ABB RAPID module: Module1.mod

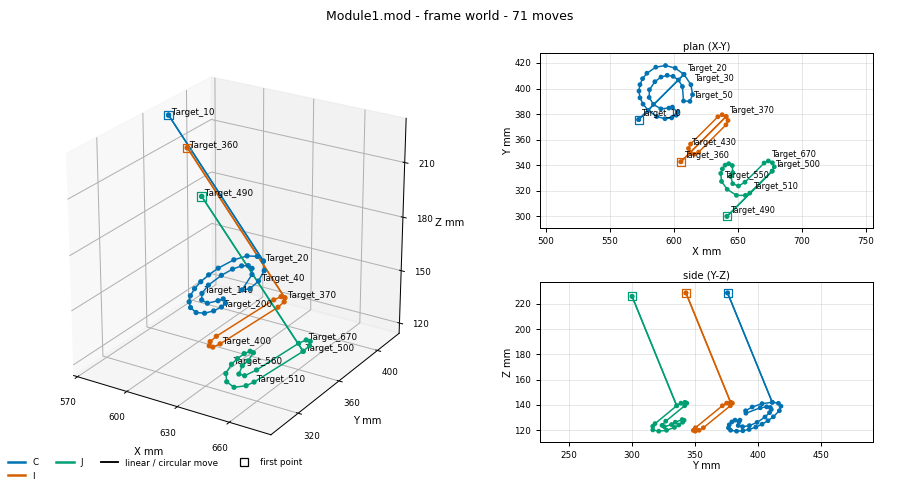
[picture p0: tool path of Module1.mod in frame world, 71 of 73 moves have a stored position in this frame; points joined in program order, loops and branches not executed]
MODULE Module1
        CONST robtarget Target_10:=[[103.793570023,149.495277511,99.999575997],[0.000000083,-0.533161025,0.846013783,0.00000013],[0,0,0,0],[9E+09,9E+09,9E+09,9E+09,9E+09,9E+09]];
    CONST robtarget Target_20:=[[103.793570137,149.495246706,-0.000424002],[0.000000083,-0.533161025,0.846013783,0.00000013],[0,0,-1,0],[9E+09,9E+09,9E+09,9E+09,9E+09,9E+09]];
    CONST robtarget Target_30:=[[113.359124829,147.348233514,-0.000423331],[0.000000133,-0.533160983,0.846013809,0.000000079],[0,0,-1,0],[9E+09,9E+09,9E+09,9E+09,9E+09,9E+09]];
    CONST robtarget Target_40:=[[119.782709001,142.041794411,-0.000421688],[0.000000153,-0.533160941,0.846013836,0.000000008],[0,0,-1,0],[9E+09,9E+09,9E+09,9E+09,9E+09,9E+09]];
    CONST robtarget Target_50:=[[122.016999147,136.089505814,-0.000419852],[-0.000000082,-0.533160946,0.846013833,-0.00000013],[0,0,-1,0],[9E+09,9E+09,9E+09,9E+09,9E+09,9E+09]];
    CONST robtarget Target_60:=[[118.316456088,132.214408841,-0.000418663],[-0.000000081,-0.533160946,0.846013833,-0.000000131],[0,0,-1,0],[9E+09,9E+09,9E+09,9E+09,9E+09,9E+09]];
    CONST robtarget Target_70:=[[109.693492554,140.750095424,-0.000421301],[-0.000000082,-0.533160946,0.846013833,-0.000000131],[0,0,-1,0],[9E+09,9E+09,9E+09,9E+09,9E+09,9E+09]];
    CONST robtarget Target_80:=[[103.863391701,142.373446861,-0.000421809],[-0.000000081,-0.533160946,0.846013833,-0.000000131],[0,0,-1,0],[9E+09,9E+09,9E+09,9E+09,9E+09,9E+09]];
    CONST robtarget Target_90:=[[98.906060436,141.326123357,-0.000421492],[-0.000000081,-0.533160946,0.846013833,-0.000000131],[0,0,-1,0],[9E+09,9E+09,9E+09,9E+09,9E+09,9E+09]];
    CONST robtarget Target_100:=[[95.065874244,138.184152838,-0.000420528],[-0.000000082,-0.533160946,0.846013833,-0.000000131],[0,0,-1,0],[9E+09,9E+09,9E+09,9E+09,9E+09,9E+09]];
    CONST robtarget Target_110:=[[92.604664001,133.104633832,-0.000418965],[-0.000000082,-0.533160946,0.846013833,-0.000000131],[0,0,-1,0],[9E+09,9E+09,9E+09,9E+09,9E+09,9E+09]];
    CONST robtarget Target_120:=[[91.784260586,126.244664864,-0.000416854],[-0.000000082,-0.533160946,0.846013833,-0.00000013],[0,0,-1,0],[9E+09,9E+09,9E+09,9E+09,9E+09,9E+09]];
    CONST robtarget Target_130:=[[93.2330581,117.656612109,-0.000414207],[0.000000152,-0.533160925,0.846013846,-0.000000026],[0,0,-1,0],[9E+09,9E+09,9E+09,9E+09,9E+09,9E+09]];
    CONST robtarget Target_140:=[[97.335075165,112.542182317,-0.000412627],[0.00000014,-0.533160974,0.846013815,0.000000065],[0,0,-1,0],[9E+09,9E+09,9E+09,9E+09,9E+09,9E+09]];
    CONST robtarget Target_150:=[[103.549194637,110.849009312,-0.000412097],[0.000000083,-0.533161025,0.846013783,0.00000013],[0,0,-1,0],[9E+09,9E+09,9E+09,9E+09,9E+09,9E+09]];
    CONST robtarget Target_160:=[[110.094966554,112.769102406,-0.000412682],[-0.000000009,-0.533161065,0.846013758,0.000000153],[0,0,-1,0],[9E+09,9E+09,9E+09,9E+09,9E+09,9E+09]];
    CONST robtarget Target_170:=[[114.127162057,118.389738556,-0.000414408],[-0.000000094,-0.533161077,0.846013751,0.000000123],[0,0,-1,0],[9E+09,9E+09,9E+09,9E+09,9E+09,9E+09]];
    CONST robtarget Target_180:=[[115.5235934,121.252422806,-0.000415289],[-0.000000055,-0.533161075,0.846013751,0.000000144],[0,0,-1,0],[9E+09,9E+09,9E+09,9E+09,9E+09,9E+09]];
    CONST robtarget Target_190:=[[120.987131026,121.252422805,-0.000415283],[0.00000015,-0.533160956,0.846013827,0.000000034],[0,0,-1,0],[9E+09,9E+09,9E+09,9E+09,9E+09,9E+09]];
    CONST robtarget Target_200:=[[122.12173149,118.45956012,-0.000414421],[-0.000000082,-0.533160946,0.846013833,-0.00000013],[0,0,-1,0],[9E+09,9E+09,9E+09,9E+09,9E+09,9E+09]];
    CONST robtarget Target_210:=[[121.091863374,113.886247475,-0.000413014],[-0.000000082,-0.533160946,0.846013833,-0.000000131],[0,0,-1,0],[9E+09,9E+09,9E+09,9E+09,9E+09,9E+09]];
    CONST robtarget Target_220:=[[117.82770511,109.068559346,-0.000411533],[-0.000000081,-0.533160946,0.846013833,-0.00000013],[0,0,-1,0],[9E+09,9E+09,9E+09,9E+09,9E+09,9E+09]];
    CONST robtarget Target_230:=[[112.119791998,105.210917765,-0.000410351],[-0.000000081,-0.533160946,0.846013833,-0.000000131],[0,0,-1,0],[9E+09,9E+09,9E+09,9E+09,9E+09,9E+09]];
    CONST robtarget Target_240:=[[104.037945604,103.727209468,-0.000409903],[-0.000000081,-0.533160946,0.846013833,-0.000000131],[0,0,-1,0],[9E+09,9E+09,9E+09,9E+09,9E+09,9E+09]];
    CONST robtarget Target_250:=[[97.666727605,104.390514357,-0.000410115],[-0.000000082,-0.533160946,0.846013833,-0.000000131],[0,0,-1,0],[9E+09,9E+09,9E+09,9E+09,9E+09,9E+09]];
    CONST robtarget Target_260:=[[92.447565465,106.450250589,-0.000410756],[-0.000000081,-0.533160946,0.846013833,-0.000000131],[0,0,-1,0],[9E+09,9E+09,9E+09,9E+09,9E+09,9E+09]];
    CONST robtarget Target_270:=[[88.15353909,110.150793647,-0.0004119],[-0.000000082,-0.533160946,0.846013833,-0.000000132],[0,0,-1,0],[9E+09,9E+09,9E+09,9E+09,9E+09,9E+09]];
    CONST robtarget Target_280:=[[85.168667098,114.828838645,-0.000413345],[-0.000000082,-0.533160947,0.846013833,-0.00000013],[0,0,-1,0],[9E+09,9E+09,9E+09,9E+09,9E+09,9E+09]];
    CONST robtarget Target_290:=[[83.318395571,120.327287055,-0.000415041],[-0.000000082,-0.533160946,0.846013833,-0.00000013],[0,0,-1,0],[9E+09,9E+09,9E+09,9E+09,9E+09,9E+09]];
    CONST robtarget Target_300:=[[82.707456862,126.558861919,-0.000416961],[-0.00000013,-0.533161068,0.846013756,0.000000082],[0,0,-1,0],[9E+09,9E+09,9E+09,9E+09,9E+09,9E+09]];
    CONST robtarget Target_310:=[[84.260986733,136.124416613,-0.000419906],[-0.000000094,-0.533161077,0.846013751,0.000000123],[0,0,-1,0],[9E+09,9E+09,9E+09,9E+09,9E+09,9E+09]];
    CONST robtarget Target_320:=[[88.712111639,143.350948806,-0.000422127],[-0.000000037,-0.533161072,0.846013754,0.000000149],[0,0,-1,0],[9E+09,9E+09,9E+09,9E+09,9E+09,9E+09]];
    CONST robtarget Target_330:=[[95.502259042,147.924261449,-0.000423527],[0.000000028,-0.533161053,0.846013766,0.000000151],[0,0,-1,0],[9E+09,9E+09,9E+09,9E+09,9E+09,9E+09]];
    CONST robtarget Target_340:=[[103.793570137,149.495246706,-0.000424002],[0.000000083,-0.533161025,0.846013783,0.00000013],[0,0,-1,0],[9E+09,9E+09,9E+09,9E+09,9E+09,9E+09]];
    CONST robtarget Target_350:=[[103.793570023,149.495277511,99.999575997],[0.000000083,-0.533161025,0.846013783,0.00000013],[0,0,-1,0],[9E+09,9E+09,9E+09,9E+09,9E+09,9E+09]];
    CONST robtarget Target_360:=[[150.434376851,149.495277492,99.999576051],[0.000000083,-0.533161025,0.846013783,0.00000013],[0,0,0,0],[9E+09,9E+09,9E+09,9E+09,9E+09,9E+09]];
    CONST robtarget Target_370:=[[150.434376963,149.495246688,-0.000423949],[0.000000083,-0.533161025,0.846013783,0.00000013],[0,0,-1,0],[9E+09,9E+09,9E+09,9E+09,9E+09,9E+09]];
    CONST robtarget Target_380:=[[153.681079834,148.15118152,-0.000423532],[0.000000151,-0.533160952,0.846013829,0.000000028],[0,0,-1,0],[9E+09,9E+09,9E+09,9E+09,9E+09,9E+09]];
    CONST robtarget Target_390:=[[154.93786804,144.049164452,-0.000422267],[-0.000000082,-0.533160946,0.846013833,-0.00000013],[0,0,-1,0],[9E+09,9E+09,9E+09,9E+09,9E+09,9E+09]];
    CONST robtarget Target_400:=[[154.937868027,109.208202466,-0.000411535],[-0.000000082,-0.533160946,0.846013833,-0.00000013],[0,0,-1,0],[9E+09,9E+09,9E+09,9E+09,9E+09,9E+09]];
    CONST robtarget Target_410:=[[153.681079818,105.088730007,-0.000410266],[-0.000000081,-0.533160946,0.846013833,-0.000000131],[0,0,-1,0],[9E+09,9E+09,9E+09,9E+09,9E+09,9E+09]];
    CONST robtarget Target_420:=[[150.434376946,103.72720945,-0.00040985],[-0.000000081,-0.533160946,0.846013833,-0.000000131],[0,0,-1,0],[9E+09,9E+09,9E+09,9E+09,9E+09,9E+09]];
    CONST robtarget Target_430:=[[147.257495644,105.106185402,-0.000410279],[-0.000000082,-0.533160946,0.846013833,-0.000000131],[0,0,-1,0],[9E+09,9E+09,9E+09,9E+09,9E+09,9E+09]];
    CONST robtarget Target_440:=[[146.000707437,109.208202469,-0.000411544],[-0.00000013,-0.533161068,0.846013756,0.000000082],[0,0,-1,0],[9E+09,9E+09,9E+09,9E+09,9E+09,9E+09]];
    CONST robtarget Target_450:=[[146.00070745,144.049164456,-0.000422278],[-0.00000013,-0.533161068,0.846013756,0.000000082],[0,0,-1,0],[9E+09,9E+09,9E+09,9E+09,9E+09,9E+09]];
    CONST robtarget Target_460:=[[147.240040268,148.13372613,-0.000423534],[-0.000000041,-0.533161073,0.846013753,0.000000149],[0,0,-1,0],[9E+09,9E+09,9E+09,9E+09,9E+09,9E+09]];
    CONST robtarget Target_470:=[[150.434376963,149.495246688,-0.000423949],[0.000000083,-0.533161025,0.846013783,0.00000013],[0,0,-1,0],[9E+09,9E+09,9E+09,9E+09,9E+09,9E+09]];
    CONST robtarget Target_480:=[[150.434376851,149.495277492,99.999576051],[0.000000083,-0.533161025,0.846013783,0.00000013],[0,0,-1,0],[9E+09,9E+09,9E+09,9E+09,9E+09,9E+09]];
    CONST robtarget Target_490:=[[206.082165832,144.049195237,99.999577791],[-0.000000082,-0.533160946,0.846013833,-0.00000013],[0,0,0,0],[9E+09,9E+09,9E+09,9E+09,9E+09,9E+09]];
    CONST robtarget Target_500:=[[206.082165946,144.049164432,-0.000422209],[-0.000000082,-0.533160946,0.846013833,-0.00000013],[0,0,-1,0],[9E+09,9E+09,9E+09,9E+09,9E+09,9E+09]];
    CONST robtarget Target_510:=[[205.820335058,115.753974363,-0.000413492],[-0.000000082,-0.533160946,0.846013833,-0.000000131],[0,0,-1,0],[9E+09,9E+09,9E+09,9E+09,9E+09,9E+09]];
    CONST robtarget Target_520:=[[204.650823807,111.442492595,-0.000412166],[-0.000000082,-0.533160947,0.846013833,-0.00000013],[0,0,-1,0],[9E+09,9E+09,9E+09,9E+09,9E+09,9E+09]];
    CONST robtarget Target_530:=[[199.69349254,105.769490269,-0.000410425],[-0.000000082,-0.533160946,0.846013833,-0.000000131],[0,0,-1,0],[9E+09,9E+09,9E+09,9E+09,9E+09,9E+09]];
    CONST robtarget Target_540:=[[191.24508292,103.727209435,-0.000409804],[-0.000000081,-0.533160946,0.846013833,-0.000000131],[0,0,-1,0],[9E+09,9E+09,9E+09,9E+09,9E+09,9E+09]];
    CONST robtarget Target_550:=[[183.77417524,105.14109617,-0.000410249],[-0.000000081,-0.533160946,0.846013833,-0.000000131],[0,0,-1,0],[9E+09,9E+09,9E+09,9E+09,9E+09,9E+09]];
    CONST robtarget Target_560:=[[178.921576328,109.731864211,-0.000411669],[-0.000000082,-0.533160946,0.846013833,-0.000000131],[0,0,-1,0],[9E+09,9E+09,9E+09,9E+09,9E+09,9E+09]];
    CONST robtarget Target_570:=[[177.35059107,113.624416577,-0.000412869],[-0.000000081,-0.533160946,0.846013833,-0.00000013],[0,0,-1,0],[9E+09,9E+09,9E+09,9E+09,9E+09,9E+09]];
    CONST robtarget Target_580:=[[176.757107751,117.831165995,-0.000414166],[-0.00000013,-0.533161068,0.846013756,0.000000082],[0,0,-1,0],[9E+09,9E+09,9E+09,9E+09,9E+09,9E+09]];
    CONST robtarget Target_590:=[[177.926619001,121.042958082,-0.000415153],[-0.00000003,-0.533161071,0.846013754,0.000000151],[0,0,-1,0],[9E+09,9E+09,9E+09,9E+09,9E+09,9E+09]];
    CONST robtarget Target_600:=[[180.946401779,122.160103154,-0.000415494],[0.000000083,-0.533161025,0.846013783,0.00000013],[0,0,-1,0],[9E+09,9E+09,9E+09,9E+09,9E+09,9E+09]];
    CONST robtarget Target_610:=[[185.030963453,117.935898343,-0.000414188],[0.000000145,-0.533160914,0.846013853,-0.000000052],[0,0,-1,0],[9E+09,9E+09,9E+09,9E+09,9E+09,9E+09]];
    CONST robtarget Target_620:=[[186.043376174,114.235355286,-0.000413048],[0.00000015,-0.533160923,0.846013848,-0.000000032],[0,0,-1,0],[9E+09,9E+09,9E+09,9E+09,9E+09,9E+09]];
    CONST robtarget Target_630:=[[191.210172139,110.849009279,-0.000411998],[0.000000083,-0.533161025,0.846013783,0.00000013],[0,0,-1,0],[9E+09,9E+09,9E+09,9E+09,9E+09,9E+09]];
    CONST robtarget Target_640:=[[195.661297043,113.03093325,-0.000412666],[-0.000000061,-0.533161076,0.846013751,0.000000141],[0,0,-1,0],[9E+09,9E+09,9E+09,9E+09,9E+09,9E+09]];
    CONST robtarget Target_650:=[[197.145005346,119.576705165,-0.00041468],[-0.00000013,-0.533161068,0.846013756,0.000000082],[0,0,-1,0],[9E+09,9E+09,9E+09,9E+09,9E+09,9E+09]];
    CONST robtarget Target_660:=[[197.145005355,144.049164436,-0.000422219],[-0.00000013,-0.533161068,0.846013756,0.000000082],[0,0,-1,0],[9E+09,9E+09,9E+09,9E+09,9E+09,9E+09]];
    CONST robtarget Target_670:=[[198.331971998,148.133726111,-0.000423476],[-0.000000043,-0.533161074,0.846013753,0.000000148],[0,0,-1,0],[9E+09,9E+09,9E+09,9E+09,9E+09,9E+09]];
    CONST robtarget Target_680:=[[201.578674869,149.495246669,-0.000423891],[0.000000083,-0.533161025,0.846013783,0.00000013],[0,0,-1,0],[9E+09,9E+09,9E+09,9E+09,9E+09,9E+09]];
    CONST robtarget Target_690:=[[204.860288522,148.133726108,-0.000423468],[0.000000152,-0.53316095,0.84601383,0.000000025],[0,0,-1,0],[9E+09,9E+09,9E+09,9E+09,9E+09,9E+09]];
    CONST robtarget Target_700:=[[206.082165946,144.049164432,-0.000422209],[-0.000000082,-0.533160946,0.846013833,-0.00000013],[0,0,-1,0],[9E+09,9E+09,9E+09,9E+09,9E+09,9E+09]];
    CONST robtarget Target_710:=[[206.082165832,144.049195237,99.999577791],[-0.000000082,-0.533160946,0.846013833,-0.00000013],[0,0,-1,0],[9E+09,9E+09,9E+09,9E+09,9E+09,9E+09]];
    CONST jointtarget Home:=[[0,0,0,0,30,0],[9E+09,9E+09,9E+09,9E+09,9E+09,9E+09]];
    CONST jointtarget Mantenimiento:=[[90,0,0,0,0,0],[9E+09,9E+09,9E+09,9E+09,9E+09,9E+09]];
!***********************************************************
    !
    ! Módulo:  Module1
    !
    ! Descripción:
    !   <Introduzca la descripción aquí>
    !
    ! Autor: Sebastián
    !
    ! Versión: 1.0
    !
    !***********************************************************


    !***********************************************************
    !
    ! Procedimiento Main
    !
    !   Este es el punto de entrada de su programa
    !
    !***********************************************************
    PROC main()
        !Añada aquí su código
        Home_;
        WaitDI Entrada1,1;
        SetDO Salida1,1;
        C;
        I;
        J;
        Home_;
        WaitDI Entrada2,1;
        SetDO Salida1,0;
        mantenimiento_;


    ENDPROC
    PROC C()
        MoveL Target_10,v100,z10,Herr_CIJ\WObj:=Tablero_CIJ;
        MoveL Target_20,v100,z10,Herr_CIJ\WObj:=Tablero_CIJ;
        MoveL Target_30,v100,z10,Herr_CIJ\WObj:=Tablero_CIJ;
        MoveL Target_40,v100,z10,Herr_CIJ\WObj:=Tablero_CIJ;
        MoveL Target_50,v100,z10,Herr_CIJ\WObj:=Tablero_CIJ;
        MoveL Target_60,v100,z10,Herr_CIJ\WObj:=Tablero_CIJ;
        MoveL Target_70,v100,z10,Herr_CIJ\WObj:=Tablero_CIJ;
        MoveL Target_80,v100,z10,Herr_CIJ\WObj:=Tablero_CIJ;
        MoveL Target_90,v100,z10,Herr_CIJ\WObj:=Tablero_CIJ;
        MoveL Target_100,v100,z10,Herr_CIJ\WObj:=Tablero_CIJ;
        MoveL Target_110,v100,z10,Herr_CIJ\WObj:=Tablero_CIJ;
        MoveL Target_120,v100,z10,Herr_CIJ\WObj:=Tablero_CIJ;
        MoveL Target_130,v100,z10,Herr_CIJ\WObj:=Tablero_CIJ;
        MoveL Target_140,v100,z10,Herr_CIJ\WObj:=Tablero_CIJ;
        MoveL Target_150,v100,z10,Herr_CIJ\WObj:=Tablero_CIJ;
        MoveL Target_160,v100,z10,Herr_CIJ\WObj:=Tablero_CIJ;
        MoveL Target_170,v100,z10,Herr_CIJ\WObj:=Tablero_CIJ;
        MoveL Target_180,v100,z10,Herr_CIJ\WObj:=Tablero_CIJ;
        MoveL Target_190,v100,z10,Herr_CIJ\WObj:=Tablero_CIJ;
        MoveL Target_200,v100,z10,Herr_CIJ\WObj:=Tablero_CIJ;
        MoveL Target_210,v100,z10,Herr_CIJ\WObj:=Tablero_CIJ;
        MoveL Target_220,v100,z10,Herr_CIJ\WObj:=Tablero_CIJ;
        MoveL Target_230,v100,z10,Herr_CIJ\WObj:=Tablero_CIJ;
        MoveL Target_240,v100,z10,Herr_CIJ\WObj:=Tablero_CIJ;
        MoveL Target_250,v100,z10,Herr_CIJ\WObj:=Tablero_CIJ;
        MoveL Target_260,v100,z10,Herr_CIJ\WObj:=Tablero_CIJ;
        MoveL Target_270,v100,z10,Herr_CIJ\WObj:=Tablero_CIJ;
        MoveL Target_280,v100,z10,Herr_CIJ\WObj:=Tablero_CIJ;
        MoveL Target_290,v100,z10,Herr_CIJ\WObj:=Tablero_CIJ;
        MoveL Target_300,v100,z10,Herr_CIJ\WObj:=Tablero_CIJ;
        MoveL Target_310,v100,z10,Herr_CIJ\WObj:=Tablero_CIJ;
        MoveL Target_320,v100,z10,Herr_CIJ\WObj:=Tablero_CIJ;
        MoveL Target_330,v100,z10,Herr_CIJ\WObj:=Tablero_CIJ;
        MoveL Target_340,v100,z10,Herr_CIJ\WObj:=Tablero_CIJ;
        MoveL Target_350,v100,z10,Herr_CIJ\WObj:=Tablero_CIJ;
    ENDPROC
    PROC I()
        MoveL Target_360,v100,z10,Herr_CIJ\WObj:=Tablero_CIJ;
        MoveL Target_370,v100,z10,Herr_CIJ\WObj:=Tablero_CIJ;
        MoveL Target_380,v100,z10,Herr_CIJ\WObj:=Tablero_CIJ;
        MoveL Target_390,v100,z10,Herr_CIJ\WObj:=Tablero_CIJ;
        MoveL Target_400,v100,z10,Herr_CIJ\WObj:=Tablero_CIJ;
        MoveL Target_410,v100,z10,Herr_CIJ\WObj:=Tablero_CIJ;
        MoveL Target_420,v100,z10,Herr_CIJ\WObj:=Tablero_CIJ;
        MoveL Target_430,v100,z10,Herr_CIJ\WObj:=Tablero_CIJ;
        MoveL Target_440,v100,z10,Herr_CIJ\WObj:=Tablero_CIJ;
        MoveL Target_450,v100,z10,Herr_CIJ\WObj:=Tablero_CIJ;
        MoveL Target_460,v100,z10,Herr_CIJ\WObj:=Tablero_CIJ;
        MoveL Target_470,v100,z10,Herr_CIJ\WObj:=Tablero_CIJ;
        MoveL Target_480,v100,z10,Herr_CIJ\WObj:=Tablero_CIJ;
    ENDPROC
    PROC J()
        MoveL Target_490,v100,z10,Herr_CIJ\WObj:=Tablero_CIJ;
        MoveL Target_500,v100,z10,Herr_CIJ\WObj:=Tablero_CIJ;
        MoveL Target_510,v100,z10,Herr_CIJ\WObj:=Tablero_CIJ;
        MoveL Target_520,v100,z10,Herr_CIJ\WObj:=Tablero_CIJ;
        MoveL Target_530,v100,z10,Herr_CIJ\WObj:=Tablero_CIJ;
        MoveL Target_540,v100,z10,Herr_CIJ\WObj:=Tablero_CIJ;
        MoveL Target_550,v100,z10,Herr_CIJ\WObj:=Tablero_CIJ;
        MoveL Target_560,v100,z10,Herr_CIJ\WObj:=Tablero_CIJ;
        MoveL Target_570,v100,z10,Herr_CIJ\WObj:=Tablero_CIJ;
        MoveL Target_580,v100,z10,Herr_CIJ\WObj:=Tablero_CIJ;
        MoveL Target_590,v100,z10,Herr_CIJ\WObj:=Tablero_CIJ;
        MoveL Target_600,v100,z10,Herr_CIJ\WObj:=Tablero_CIJ;
        MoveL Target_610,v100,z10,Herr_CIJ\WObj:=Tablero_CIJ;
        MoveL Target_620,v100,z10,Herr_CIJ\WObj:=Tablero_CIJ;
        MoveL Target_630,v100,z10,Herr_CIJ\WObj:=Tablero_CIJ;
        MoveL Target_640,v100,z10,Herr_CIJ\WObj:=Tablero_CIJ;
        MoveL Target_650,v100,z10,Herr_CIJ\WObj:=Tablero_CIJ;
        MoveL Target_660,v100,z10,Herr_CIJ\WObj:=Tablero_CIJ;
        MoveL Target_670,v100,z10,Herr_CIJ\WObj:=Tablero_CIJ;
        MoveL Target_680,v100,z10,Herr_CIJ\WObj:=Tablero_CIJ;
        MoveL Target_690,v100,z10,Herr_CIJ\WObj:=Tablero_CIJ;
        MoveL Target_700,v100,z10,Herr_CIJ\WObj:=Tablero_CIJ;
        MoveL Target_710,v100,z10,Herr_CIJ\WObj:=Tablero_CIJ;
    ENDPROC
    PROC Home_()
        MoveAbsJ Home,v1000,z100,Herr_CIJ\WObj:=Tablero_CIJ;
    ENDPROC
    PROC mantenimiento_()
        MoveAbsJ Mantenimiento,v1000,z100,Herr_CIJ\WObj:=Tablero_CIJ;
    ENDPROC
ENDMODULE
